PROGRAM MAIN
VAR
END_VAR

PRG_Thermocouple();
PRG_PowerMeasurement();
PRG_MotorDrive();
PRG_VfdModbusRtu();

END_PROGRAM

(* stored: Version 1.1.0.1, ProductVersion 3.1.4024.12
   POU MAIN: Id {a7a66e3d-c8d9-4253-86bf-86db8e9c4fd5}, SpecialFunc None *)
